(* PLC project SafeLOGIC-1, BrAutomation SafeDESIGNER  4.3.4.4 *)
(* stored: companyURL http://www.br-automation.com, creationDateTime Fri Oct 19 12:00:31 2018 *)

PROGRAM GuardLocks

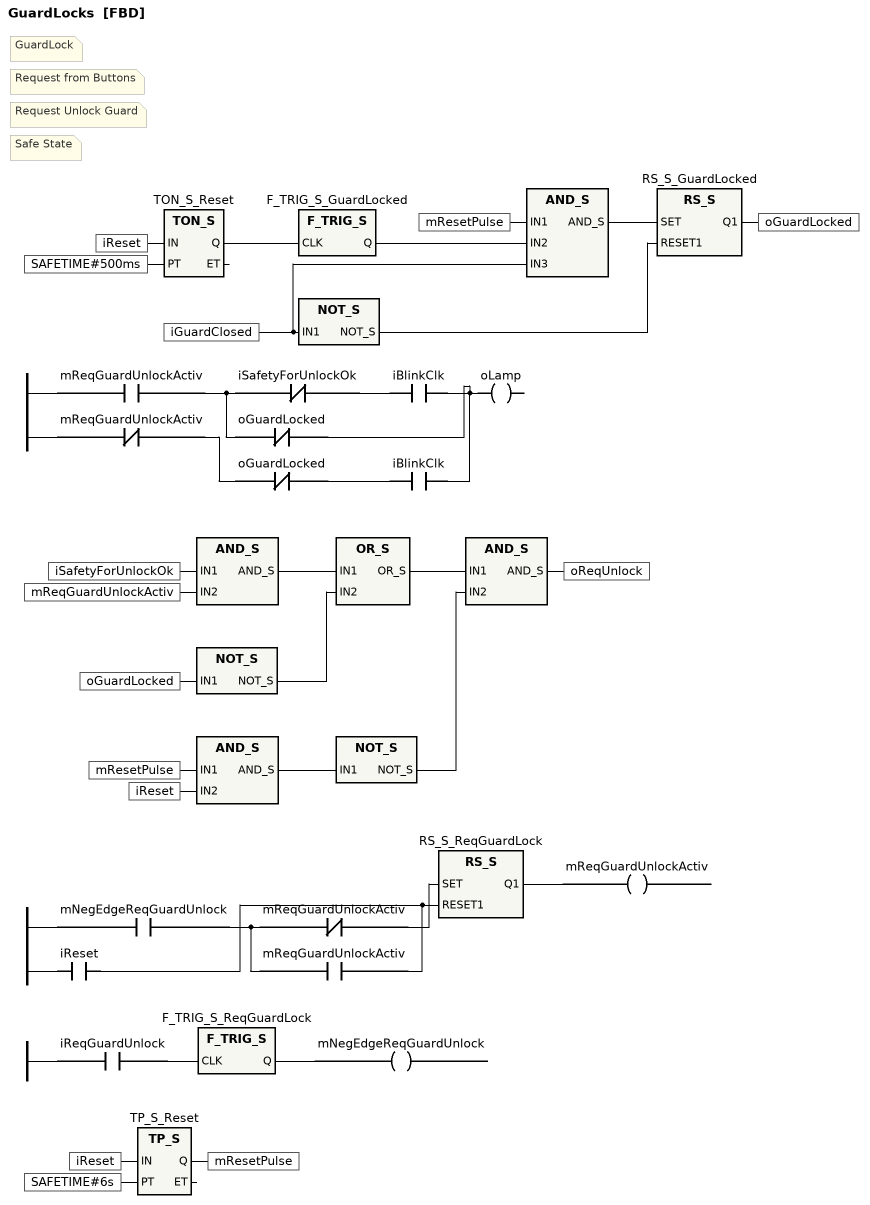
(* FBD diagram, written out as Structured Text *)
(* GuardLock *)
(* Request from Buttons *)
F_TRIG_S_ReqGuardLock(CLK := iReqGuardUnlock);
mNegEdgeReqGuardUnlock := F_TRIG_S_ReqGuardLock.Q;
RS_S_ReqGuardLock(SET := mNegEdgeReqGuardUnlock AND NOT mReqGuardUnlockActiv, RESET1 := mNegEdgeReqGuardUnlock AND mReqGuardUnlockActiv OR iReset);
mReqGuardUnlockActiv := RS_S_ReqGuardLock.Q1;
TP_S_Reset(IN := iReset, PT := SAFETIME#6s);
mResetPulse := TP_S_Reset.Q;
(* Safe State *)
TON_S_Reset(IN := iReset, PT := SAFETIME#500ms);
F_TRIG_S_GuardLocked(CLK := TON_S_Reset.Q);
RS_S_GuardLocked(SET := AND_S(mResetPulse, F_TRIG_S_GuardLocked.Q, iGuardClosed), RESET1 := NOT_S(iGuardClosed));
oGuardLocked := RS_S_GuardLocked.Q1;
(* Request Unlock Guard *)
oReqUnlock := AND_S(OR_S(AND_S(iSafetyForUnlockOk, mReqGuardUnlockActiv), NOT_S(oGuardLocked)), NOT_S(AND_S(mResetPulse, iReset)));
oLamp := mReqGuardUnlockActiv AND NOT iSafetyForUnlockOk AND iBlinkClk OR mReqGuardUnlockActiv AND NOT oGuardLocked OR NOT mReqGuardUnlockActiv AND NOT oGuardLocked AND iBlinkClk;
END_PROGRAM
